// TIA Portal V17 export
// export: Created 2026-04-13T11:12:44.8442208Z, ExportSetting WithDefaults, DisplayName Totally Integrated Automation Portal, DisplayVersion V17 Update 4, DisplayName TIA Portal Openness, DisplayVersion V17 Update 4, DisplayName TIA Portal Version Control Interface, DisplayVersion V17, DisplayName SINAMICS Startdrive Advanced, DisplayVersion V17, DisplayName SINAMICS Startdrive G130, G150, S120, S150, SINAMICS MV, S210, DisplayVersion V17, DisplayName SINAMICS Startdrive G110M, G120, G120C, G120D, G120P, G115D, DisplayVersion V17, DisplayName STEP 7 Professional, DisplayVersion V17 Update 4, DisplayName STEP 7 Safety, DisplayVersion V17, DisplayName WinCC Professional, DisplayVersion V17 Update 4
FUNCTION "GetSymbolName" : WString   // FC910, SCL
TITLE = GetSymbolName
AUTHOR : Siemens
FAMILY : SymInfo
NAME : GetSymNa
VERSION : 1.2
// stored: IsIECCheckEnabled false, SetENOAutomatically false, UDAEnableTagReadback false
   VAR_INPUT
      SymInfo : Variant;
      ParaNr : UInt;
      Size : DInt;
   END_VAR
BEGIN
END_FUNCTION
